FUNCTION_BLOCK FB_Skill EXTENDS FB_Base IMPLEMENTS  ITF_1_Skill
VAR_INPUT
	SFCInit, SFCPause, SFCReset: BOOL;
END_VAR
VAR_OUTPUT
	bBusy, bDone: BOOL;
	SFCError: BOOL;
	SFCCurrentStep: STRING;
END_VAR
VAR
	SubSkillHandler : FB_SkillHandler;
END_VAR

{warning 'Add method implementation '}
METHOD M_Pause : BOOL
IF _state=eState.Active THEN
	SFCPause:=TRUE;
END_IF
END_METHOD

{warning 'Add method implementation '}
METHOD M_Restart : BOOL //Stay activ, but restart
SFCReset:=True;
END_METHOD

{warning 'Add method implementation '}
METHOD M_Resume : BOOL
SFCPause:=False;
END_METHOD

{warning 'Add method implementation '}
METHOD M_Start : BOOL
M_activate();
END_METHOD

{warning 'Add method implementation '}
METHOD M_Stop : BOOL
IF _state=eState.Active THEN
	SFCPause:=TRUE;
	M_deactivate();
END_IF
END_METHOD

METHOD onActivate : BOOL
// ---- Init ----
transitionresult:=eResult.None;



// ---- Change ----




// ---- Check ----
transitionresult := eResult.SUCCESS;


// ---- Change State ----
IF transitionresult= eResult.SUCCESS THEN
	P_State:=eState.Active;
ELSIF transitionresult= eResult.FAILURE THEN
	P_State:=eState.Inactive;
ELSIF transitionresult= eResult.ERROR THEN
	P_State:=eState.ErrorProcessing;
ELSE
	ADSLOGSTR(ADSLOG_MSGTYPE_WARN,'Transitionresult from onActivate is None','');
END_IF
END_METHOD

METHOD onCleanup : BOOL
// ---- Init ----
transitionresult:=eResult.None;



// ---- Change ----



// ---- Check ----
transitionresult := eResult.SUCCESS;


// ---- Change State ----
IF transitionresult= eResult.SUCCESS THEN
	P_State:=eState.Unconfigured;
ELSIF transitionresult= eResult.FAILURE THEN
	ADSLOGSTR(ADSLOG_MSGTYPE_WARN,'Transitionresult from onCleanup is FAILURE ','');
ELSIF transitionresult= eResult.ERROR THEN
	P_State:=eState.ErrorProcessing;
ELSE
	ADSLOGSTR(ADSLOG_MSGTYPE_WARN,'Transitionresult from onCleanup is NONE','');
END_IF
END_METHOD

METHOD onConfigure : BOOL
// ---- Init ----
transitionresult:=eResult.None;



// ---- Change ----


// ---- Check ----
transitionresult := eResult.SUCCESS;


// ---- Change State ----
IF transitionresult= eResult.SUCCESS THEN
	P_State:=eState.Inactive;
ELSIF transitionresult= eResult.FAILURE THEN
	P_State:=eState.Unconfigured;
ELSIF transitionresult= eResult.ERROR THEN
	P_State:=eState.ErrorProcessing;
ELSE
	ADSLOGSTR(ADSLOG_MSGTYPE_WARN,'Transitionresult from onConfigure is None','');
END_IF
END_METHOD

METHOD onDeactivate : BOOL
// ---- Init ----
transitionresult:=eResult.None;



// ---- Change ----
 //Stopping SFC



// ---- Check ----
transitionresult := eResult.SUCCESS;


// ---- Change State ----
IF transitionresult= eResult.SUCCESS THEN
	P_State:=eState.Inactive;
ELSIF transitionresult= eResult.FAILURE THEN
	ADSLOGSTR(ADSLOG_MSGTYPE_WARN,'Transitionresult from onDeactivate is FAILURE','');
ELSIF transitionresult= eResult.ERROR THEN
	P_State:=eState.ErrorProcessing;
ELSE
	ADSLOGSTR(ADSLOG_MSGTYPE_WARN,'Transitionresult from onDeactivate is None','');
END_IF
END_METHOD

METHOD onError : BOOL
// ---- Init ----
transitionresult:=eResult.None;



// ---- Change ----





// ---- Check ----
transitionresult := eResult.SUCCESS;


// ---- Change State ----
IF transitionresult= eResult.SUCCESS THEN
	P_State:=eState.Unconfigured;
ELSIF transitionresult= eResult.FAILURE THEN
	P_State:=eState.Finalized;
ELSIF transitionresult= eResult.ERROR THEN
	ADSLOGSTR(ADSLOG_MSGTYPE_WARN,'Transitionresult from onError is Error','');
ELSE
	ADSLOGSTR(ADSLOG_MSGTYPE_WARN,'Transitionresult from onError is None','');
END_IF
END_METHOD

METHOD onShutdown : BOOL
// ---- Init ----
transitionresult:=eResult.None;



// ---- Change ----




// ---- Check ----
transitionresult := eResult.SUCCESS;


// ---- Change State ----
IF transitionresult= eResult.SUCCESS THEN
	P_State:=eState.Finalized;
ELSIF transitionresult= eResult.FAILURE THEN
	ADSLOGSTR(ADSLOG_MSGTYPE_WARN,'Transitionresult from onShutdown is FAILURE','');
ELSIF transitionresult= eResult.ERROR THEN
	P_State:=eState.ErrorProcessing;
ELSE
	ADSLOGSTR(ADSLOG_MSGTYPE_WARN,'Transitionresult from onShutdown is None','');
END_IF
END_METHOD

{warning 'Add property implementation'}
PROPERTY P_Busy : BOOL
GET
IF _state=eState.Active THEN
	P_Busy:=TRUE;
ELSE
	P_Busy:=FALSE;
END_IF
END_GET
END_PROPERTY

{warning 'Add property implementation'}
PROPERTY P_Done : BOOL
GET
P_Done:=bDone;
END_GET
END_PROPERTY

END_FUNCTION_BLOCK

(* stored: Version 1.1.0.1, ProductVersion 3.1.4026.18
   POU FB_Skill: Id {0b17e4be-d439-430e-8e7f-2b34d1533bf7}, SpecialFunc None
   Folder StateControl: Id {5d1d34f6-b00b-4bfe-850d-2a50e71c6867}
   Method M_Pause: Id {e320d6b1-061b-4245-81c0-f7677aa19eb4}
   Method M_Restart: Id {f7d1bc69-7e9d-4355-b12f-7afa81e0ef82}
   Method M_Resume: Id {4ac603da-7c96-44c8-afc9-9dcc8e144514}
   Method M_Start: Id {0b22be9d-d5e9-4610-815a-61f31c72ebb7}
   Method M_Stop: Id {242e45b0-6e21-4202-8089-05c40a453c9c}
   Method onActivate: Id {b6600df7-e52f-4259-bf22-90fd6ff888b9}
   Method onCleanup: Id {8f1a4b78-b2bc-40d7-b697-da534fd113b1}
   Method onConfigure: Id {cb7bdeed-2be8-42fd-bd76-167dbfd75158}
   Method onDeactivate: Id {b927a409-2ad9-49da-9542-5009ba100783}
   Method onError: Id {564f1db2-c809-4fde-b8c3-99cfbd2773f5}
   Method onShutdown: Id {ec1e4358-8bda-4b5f-a8bf-6122c7053764}
   Property P_Busy: Id {44811af8-7ac9-4c33-9fee-4ed9763a80fd}
   Get Get: Id {1acaadd8-f3a0-478f-a40d-85dfefdf6bbe}
   Property P_Done: Id {398629ef-6f21-4eea-9d45-557264c66965}
   Get Get: Id {cdfc4ba6-20c2-4e87-b8a4-7b51c8cf88bc} *)
